# EPICS autosave request: acsMotionApp/Db/SPiiPlusHoming_settings.req
$(P)$(M):homingMethod.VAL
$(P)$(M):homingMaxDist.VAL
$(P)$(M):homingOffsetPos.VAL
$(P)$(M):homingOffsetNeg.VAL
$(P)$(M):homingCurrLimit.VAL
